// TIA Portal V19 export
FUNCTION_BLOCK "A0303_Sollevamento_FB"   // FB87, LAD
// stored: MemoryReserve 100, SetENOAutomatically false
   VAR_INPUT
      AreaInterface : "AreaInterface";
      ZSI : "udt_ZoneSafetyInterface";
      DSI_Feed_Testa : "udt_DeviceSafetyInterface";
      DSI_Feed_Coda : "udt_DeviceSafetyInterface";
      DataIn : Struct
         OP_Vai_A_Prelievo : Bool;
         OP_Vai_A_Deposito : Bool;
         LsSensor1_Carico : Bool;   // FTC 1 CONTROLLO POSIZIONE LIBERA IN CARICO
         LsSensor2_Carico : Bool;   // FTC 2 CONTROLLO POSIZIONE LIBERA IN CARICO
         LsSensor1_Scarico : Bool;   // FTC 1 CONTROLLO POSIZIONE LIBERA IN SCARICO
         LsSensor2_Scarico : Bool;   // FTC 2 CONTROLLO POSIZIONE LIBERA IN SCARICO
      END_STRUCT;
      CIn : Struct
         Manager : Struct
            EnableStopDoorOpeningReq : Bool;
            EnableStopInPhase : Bool;
            EnableStopProgrammed : Bool;
            Control_ON : Bool;
            CanMoveFreely : Bool;
            TargetPosition : LReal;
            Phase : Struct
               VAI_A_PRELIEVO : Bool;
               VAI_A_PRE_DEPOSITO : Bool;
               VAI_A_DEPOSITO : Bool;
            END_STRUCT;
         END_STRUCT;
         Trasporto : Struct
            IsMeasuring : Bool;
         END_STRUCT;
      END_STRUCT;
      Config : Struct
         Testa : Struct
            Ax : "Positioning_DOL_Machine_Config";
         END_STRUCT;
         Coda : Struct
            Ax : "Positioning_DOL_Machine_Config";
         END_STRUCT;
         DelayMissingCondition { ExternalAccessible := 'False'; ExternalVisible := 'False'; ExternalWritable := 'False'} : Time := T#0MS;
      END_STRUCT;
   END_VAR
   VAR_OUTPUT
      MachineInterface : "MachineInterface";
      COut : Struct
         Ax_Testa : "Positioning_DOL_Machine_COut";
         Ax_Coda : "Positioning_DOL_Machine_COut";
         Standstill : Bool;
         Minus_CheckNext : Bool;
         Plus_CheckNext : Bool;
         Minus_Running : Bool;
         Plus_Running : Bool;
      END_STRUCT;
   END_VAR
   VAR_IN_OUT
      Par : Struct
         Ax_Man : "Positioning_DOL_Machine_Par";
         Ax_Testa_Pers : "Positioning_DOL_Machine_Pers_Data";
         Ax_Coda_Pers : "Positioning_DOL_Machine_Pers_Data";
         Enc : Struct
            Testa : "PosFbk_RTN";
            Coda : "PosFbk_RTN";
         END_STRUCT;
      END_STRUCT;
      Par_Mach : Struct
         PosDeposito : LReal;
         OffsetPrelievo : LReal;
         ToleranceWindow : LReal;
      END_STRUCT;
   END_VAR
   VAR
      Alarm : Struct
         Testa : Struct
            Ax : "Positioning_DOL_Machine_Alr";
            Enc { S7_SetPoint := 'True'} : "PosFbk_Encoder_Alr";
         END_STRUCT;
         Coda : Struct
            Ax : "Positioning_DOL_Machine_Alr";
            Enc { S7_SetPoint := 'True'} : "PosFbk_Encoder_Alr";
         END_STRUCT;
         CheckBothAxMove : Bool;
      END_STRUCT;
      Warning : Struct
         Testa : Struct
            Ax { S7_SetPoint := 'True'} : "Positioning_DOL_Machine_Wng";
         END_STRUCT;
         Coda : Struct
            Ax { S7_SetPoint := 'True'} : "Positioning_DOL_Machine_Wng";
         END_STRUCT;
         MissingCnd : Struct
            OP_VAI_A_PRELIEVO : Bool;   // Mancanza consenso lavoro
            OP_VAI_A_DEPOSITO : Bool;   // Mancanza consenso lavoro
         END_STRUCT;
      END_STRUCT;
      HMI : Struct
         Selection : Struct
            Ax : Int;   // 0= BOTH ; 1= HEAD ; 2= TAIL
         END_STRUCT;
         Testa : Struct
            PbPreset : Bool;
            PresetValue : LReal;
         END_STRUCT;
         Coda : Struct
            PbPreset : Bool;
            PresetValue : LReal;
         END_STRUCT;
         PositionGraph : Int;
      END_STRUCT;
      Sts : Struct
         OP_CanMoveFreely : Bool;
         OP_Vai_A_Prelievo_Cnd : Bool;
         OP_Vai_A_Deposito_Cnd : Bool;
         OP_Vai_A_PreDeposito_Cnd : Bool;
         Coda_PermessoDaSynchOk : Bool;
         Testa_PermessoDaSynchOk : Bool;
      END_STRUCT;
      Ctrl : Struct
         Man : Struct
            OP_Vai_A_Prelievo : Bool;
            OP_Vai_A_Deposito : Bool;
         END_STRUCT;
         Aut : Struct
            OP_Vai_A_Prelievo : Bool;
            OP_Vai_A_Deposito : Bool;
            OP_Vai_A_PreDeposito : Bool;
         END_STRUCT;
         OP_Vai_A_Prelievo : Bool;
         OP_Vai_A_Deposito : Bool;
         OP_Vai_A_PreDeposito : Bool;
      END_STRUCT;
      Ax_Testa { S7_SetPoint := 'True'} : "Positioning_DOL_Machine_FB";
      Ax_Coda { S7_SetPoint := 'True'} : "Positioning_DOL_Machine_FB";
      Enc_Testa : "PosFbk_SickAFM60";
      Enc_Testa_ITF : "PosFbk_ITF";
      Enc_Coda : "PosFbk_SickAFM60";
      Enc_Coda_ITF : "PosFbk_ITF";
      AUX { ExternalAccessible := 'False'; ExternalVisible := 'False'; ExternalWritable := 'False'} : Struct
         OP_Vai_A_Prelievo : Bool;
         OP_Vai_A_Deposito : Bool;
      END_STRUCT;
      TON_OP_VAI_A_PRELIEVO_MissingCnd : IEC_TIMER;
      TON_OP_VAI_A_DEPOSITO_MissingCnd : IEC_TIMER;
      TON_CheckAxMove { S7_SetPoint := 'True'} : IEC_TIMER;
      TON_CheckAxis { S7_SetPoint := 'True'} : IEC_TIMER;
      CheckAxisSynch { S7_SetPoint := 'True'} : "CheckAxisSynch";
      Sts_PosAxis { S7_SetPoint := 'True'} : Int;
   END_VAR
   VAR_TEMP
      PE : Struct
         OP_Vai_A_Prelievo : Bool;
         OP_Vai_A_Deposito : Bool;
      END_STRUCT;
      PosDiff : LReal;
      Axis_Testa_Behind : Bool;
      Axis_Coda_Behind : Bool;
      ValueIn : LReal;
      X1 : LReal;
      X2 : LReal;
      Ret_Val : LReal;
   END_VAR
   VAR CONSTANT
      MaxDistance : LReal := 5.0;
      MinDistance : LReal := 0.5;   // soglia inferiore per isteresi
   END_VAR
   // Config.Testa.Ax.DelayMissingCondition := T#3S;
   // Config.Testa.Ax.CyclicOBTime_ms := 10.0;
   // Config.Testa.Ax.Ax.limitMinus := 0.0;
   // Config.Testa.Ax.Ax.limitPlus := 476.0;
   // Config.Testa.Ax.Ax.Backlash := 0.0;
   // Config.Testa.Ax.Ax.BacklashActivation := FALSE;
   // Config.Testa.Ax.Ax.ToleranceWindow := 0.1;
   // Config.Testa.Ax.Ax.ToleranceWindowDelay := T#100MS;
   // Config.Testa.Ax.Ax.PreCutOff := 0.0;
   // Config.Testa.Ax.Ax.PreEndLowSpeed := 0.0;
   // Config.Testa.Ax.Ax.PreEndMedSpeed := 0.0;
   // Config.Testa.Ax.Ax.ChangeDirectionDelay := T#0MS;
   // Config.Testa.Ax.Ax.StandstillVelocity := 0.5;
   // Config.Testa.Ax.Ax.StandStillDelay := T#100MS;
   // Config.Testa.Ax.Ax.HomingDirection := FALSE;
   // Config.Testa.Ax.Ax.RecallTime := 0.0;
   // Config.Testa.Ax.Ax.VelocityFilter_T := 10.0;
   // Config.Testa.Ax.Ax.VelocityMeasUnit := 2;
   // Config.Testa.Ax.Ax.PosFbkDisabled := FALSE;
   // Config.Testa.Ax.Ax.FbkCtrlDisabled := TRUE;
   // Config.Testa.Ax.Ax_UM2."m" := 1.0;
   // Config.Testa.Ax.Ax_UM2.q := 0.0;
   // Config.Testa.Ax.S120.SpeedMotor.ReferenceVelocity := 2000.0;
   // Config.Testa.Ax.S120.SpeedMotor.InvertDirection := FALSE;
   // Config.Testa.Ax.S120.PowerOffDelay := T#5S;
   // Config.Testa.Ax.S120.StandstillVelocity := 50.0;
   // Config.Testa.Ax.S120.AccTime := 0.25;
   // Config.Testa.Ax.S120.DecTime := 0.25;
   // Config.Testa.Ax.Fan.Presence := FALSE;
   // Config.Testa.Ax.Fan.DelayOff := T#10M;
   // Config.Testa.Ax.Brake_Presence := FALSE;
   // Config.Coda.Ax.DelayMissingCondition := T#3S;
   // Config.Coda.Ax.CyclicOBTime_ms := 10.0;
   // Config.Coda.Ax.Ax.limitMinus := 0.0;
   // Config.Coda.Ax.Ax.limitPlus := 476.0;
   // Config.Coda.Ax.Ax.Backlash := 0.0;
   // Config.Coda.Ax.Ax.BacklashActivation := FALSE;
   // Config.Coda.Ax.Ax.ToleranceWindow := 0.1;
   // Config.Coda.Ax.Ax.ToleranceWindowDelay := T#100MS;
   // Config.Coda.Ax.Ax.PreCutOff := 0.0;
   // Config.Coda.Ax.Ax.PreEndLowSpeed := 0.0;
   // Config.Coda.Ax.Ax.PreEndMedSpeed := 0.0;
   // Config.Coda.Ax.Ax.ChangeDirectionDelay := T#0MS;
   // Config.Coda.Ax.Ax.StandstillVelocity := 0.5;
   // Config.Coda.Ax.Ax.StandStillDelay := T#100MS;
   // Config.Coda.Ax.Ax.HomingDirection := FALSE;
   // Config.Coda.Ax.Ax.RecallTime := 0.0;
   // Config.Coda.Ax.Ax.VelocityFilter_T := 10.0;
   // Config.Coda.Ax.Ax.VelocityMeasUnit := 2;
   // Config.Coda.Ax.Ax.PosFbkDisabled := FALSE;
   // Config.Coda.Ax.Ax.FbkCtrlDisabled := TRUE;
   // Config.Coda.Ax.Ax_UM2."m" := 1.0;
   // Config.Coda.Ax.Ax_UM2.q := 0.0;
   // Config.Coda.Ax.S120.SpeedMotor.ReferenceVelocity := 2000.0;
   // Config.Coda.Ax.S120.SpeedMotor.InvertDirection := FALSE;
   // Config.Coda.Ax.S120.PowerOffDelay := T#5S;
   // Config.Coda.Ax.S120.StandstillVelocity := 50.0;
   // Config.Coda.Ax.S120.AccTime := 0.25;
   // Config.Coda.Ax.S120.DecTime := 0.25;
   // Config.Coda.Ax.Fan.Presence := FALSE;
   // Config.Coda.Ax.Fan.DelayOff := T#10M;
   // Config.Coda.Ax.Brake_Presence := FALSE;
   VAR_TEMP   // added for the SCL form of the ladder/FBD networks
      _w1 : Bool;
   END_VAR
BEGIN

REGION Network 1 (SCL): Reset allarmi
   IF #AreaInterface.RstAlarms THEN
       #Alarm.CheckBothAxMove := FALSE;
   END_IF;
END_REGION

REGION Network 2: <+>
END_REGION

REGION Network 3: <<<<<<<<<<<<<<<<<<< OPERAZIONI >>>>>>>>>>>>>>>>>>>>>>>>
END_REGION

REGION Network 4: Operazione può muoversi liberamente perchè non sposta nessun BEAM
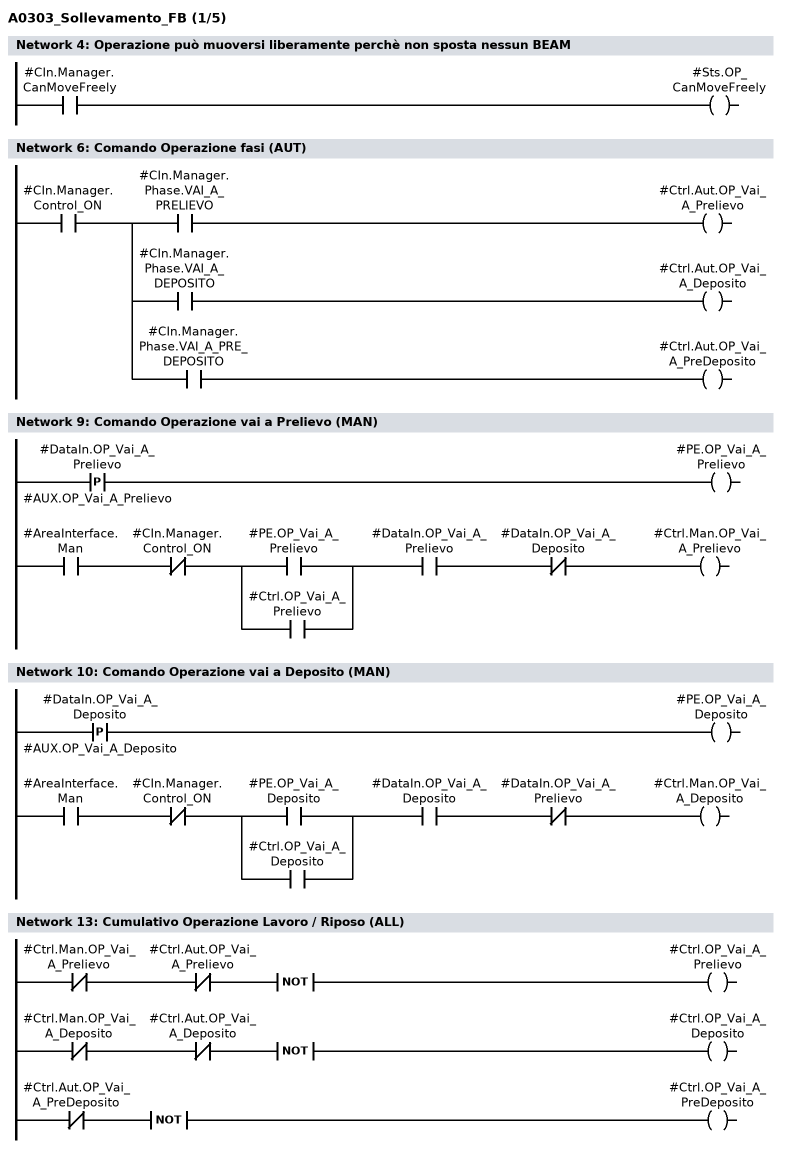
   RUNG wire#powerrail
      Contact( #CIn.Manager.CanMoveFreely )
      Coil( #Sts.OP_CanMoveFreely )
   END_RUNG
   // the same network as SCL:
   #Sts.OP_CanMoveFreely := #CIn.Manager.CanMoveFreely;
END_REGION

REGION Network 5: < OPERAZIONI AUTOMATICO >
END_REGION

REGION Network 6: Comando Operazione fasi (AUT)
   RUNG wire#powerrail
      Contact( #CIn.Manager.Control_ON )
      wire#w1
      Contact( #CIn.Manager.Phase.VAI_A_PRELIEVO )
      Coil( #Ctrl.Aut.OP_Vai_A_Prelievo )
   END_RUNG
   RUNG wire#w1
      Contact( #CIn.Manager.Phase.VAI_A_DEPOSITO )
      Coil( #Ctrl.Aut.OP_Vai_A_Deposito )
   END_RUNG
   RUNG wire#w1
      Contact( #CIn.Manager.Phase.VAI_A_PRE_DEPOSITO )
      Coil( #Ctrl.Aut.OP_Vai_A_PreDeposito )
   END_RUNG
   // the same network as SCL:
   #Ctrl.Aut.OP_Vai_A_Prelievo := #CIn.Manager.Control_ON AND #CIn.Manager.Phase.VAI_A_PRELIEVO;
   #Ctrl.Aut.OP_Vai_A_Deposito := #CIn.Manager.Control_ON AND #CIn.Manager.Phase.VAI_A_DEPOSITO;
   #Ctrl.Aut.OP_Vai_A_PreDeposito := #CIn.Manager.Control_ON AND #CIn.Manager.Phase.VAI_A_PRE_DEPOSITO;
END_REGION

REGION Network 7: <+>
END_REGION

REGION Network 8: < OPERAZIONI MANUALI >
END_REGION

REGION Network 9: Comando Operazione vai a Prelievo (MAN)
   RUNG wire#powerrail
      P_Contact(operand := #DataIn.OP_Vai_A_Prelievo, bit := #AUX.OP_Vai_A_Prelievo)
      Coil( #PE.OP_Vai_A_Prelievo )
   END_RUNG
   RUNG wire#powerrail
      Contact( #AreaInterface.Man )
      I_Contact( #CIn.Manager.Control_ON )
      wire#w1
      Contact( #PE.OP_Vai_A_Prelievo )
      wire#w2
      Contact( #DataIn.OP_Vai_A_Prelievo )
      I_Contact( #DataIn.OP_Vai_A_Deposito )
      Coil( #Ctrl.Man.OP_Vai_A_Prelievo )
   END_RUNG
   RUNG wire#w1
      Contact( #Ctrl.OP_Vai_A_Prelievo )
   END_RUNG wire#w2
   // the same network as SCL:
   #_w1 := #DataIn.OP_Vai_A_Prelievo AND NOT #AUX.OP_Vai_A_Prelievo;   // rising edge of #DataIn.OP_Vai_A_Prelievo
   #AUX.OP_Vai_A_Prelievo := #DataIn.OP_Vai_A_Prelievo;
   #PE.OP_Vai_A_Prelievo := #_w1;
   #Ctrl.Man.OP_Vai_A_Prelievo := #AreaInterface.Man AND NOT #CIn.Manager.Control_ON AND (#PE.OP_Vai_A_Prelievo OR #Ctrl.OP_Vai_A_Prelievo) AND #DataIn.OP_Vai_A_Prelievo AND NOT #DataIn.OP_Vai_A_Deposito;
END_REGION

REGION Network 10: Comando Operazione vai a Deposito (MAN)
   RUNG wire#powerrail
      P_Contact(operand := #DataIn.OP_Vai_A_Deposito, bit := #AUX.OP_Vai_A_Deposito)
      Coil( #PE.OP_Vai_A_Deposito )
   END_RUNG
   RUNG wire#powerrail
      Contact( #AreaInterface.Man )
      I_Contact( #CIn.Manager.Control_ON )
      wire#w1
      Contact( #PE.OP_Vai_A_Deposito )
      wire#w2
      Contact( #DataIn.OP_Vai_A_Deposito )
      I_Contact( #DataIn.OP_Vai_A_Prelievo )
      Coil( #Ctrl.Man.OP_Vai_A_Deposito )
   END_RUNG
   RUNG wire#w1
      Contact( #Ctrl.OP_Vai_A_Deposito )
   END_RUNG wire#w2
   // the same network as SCL:
   #_w1 := #DataIn.OP_Vai_A_Deposito AND NOT #AUX.OP_Vai_A_Deposito;   // rising edge of #DataIn.OP_Vai_A_Deposito
   #AUX.OP_Vai_A_Deposito := #DataIn.OP_Vai_A_Deposito;
   #PE.OP_Vai_A_Deposito := #_w1;
   #Ctrl.Man.OP_Vai_A_Deposito := #AreaInterface.Man AND NOT #CIn.Manager.Control_ON AND (#PE.OP_Vai_A_Deposito OR #Ctrl.OP_Vai_A_Deposito) AND #DataIn.OP_Vai_A_Deposito AND NOT #DataIn.OP_Vai_A_Prelievo;
END_REGION

REGION Network 11: <+>
END_REGION

REGION Network 12: < CUMULATIVO OPERAZIONI >
END_REGION

REGION Network 13: Cumulativo Operazione Lavoro / Riposo (ALL)
   RUNG wire#powerrail
      I_Contact( #Ctrl.Man.OP_Vai_A_Prelievo )
      I_Contact( #Ctrl.Aut.OP_Vai_A_Prelievo )
      Not()
      Coil( #Ctrl.OP_Vai_A_Prelievo )
   END_RUNG
   RUNG wire#powerrail
      I_Contact( #Ctrl.Man.OP_Vai_A_Deposito )
      I_Contact( #Ctrl.Aut.OP_Vai_A_Deposito )
      Not()
      Coil( #Ctrl.OP_Vai_A_Deposito )
   END_RUNG
   RUNG wire#powerrail
      I_Contact( #Ctrl.Aut.OP_Vai_A_PreDeposito )
      Not()
      Coil( #Ctrl.OP_Vai_A_PreDeposito )
   END_RUNG
   // the same network as SCL:
   #Ctrl.OP_Vai_A_Prelievo := NOT (NOT #Ctrl.Man.OP_Vai_A_Prelievo AND NOT #Ctrl.Aut.OP_Vai_A_Prelievo);
   #Ctrl.OP_Vai_A_Deposito := NOT (NOT #Ctrl.Man.OP_Vai_A_Deposito AND NOT #Ctrl.Aut.OP_Vai_A_Deposito);
   #Ctrl.OP_Vai_A_PreDeposito := NOT (NOT #Ctrl.Aut.OP_Vai_A_PreDeposito);
END_REGION

REGION Network 14: <+>
END_REGION

REGION Network 15: < CONDIZIONI MOVIMENTO >
END_REGION

REGION Network 16: Condizioni movimento Operazione a Lavoro / Riposo
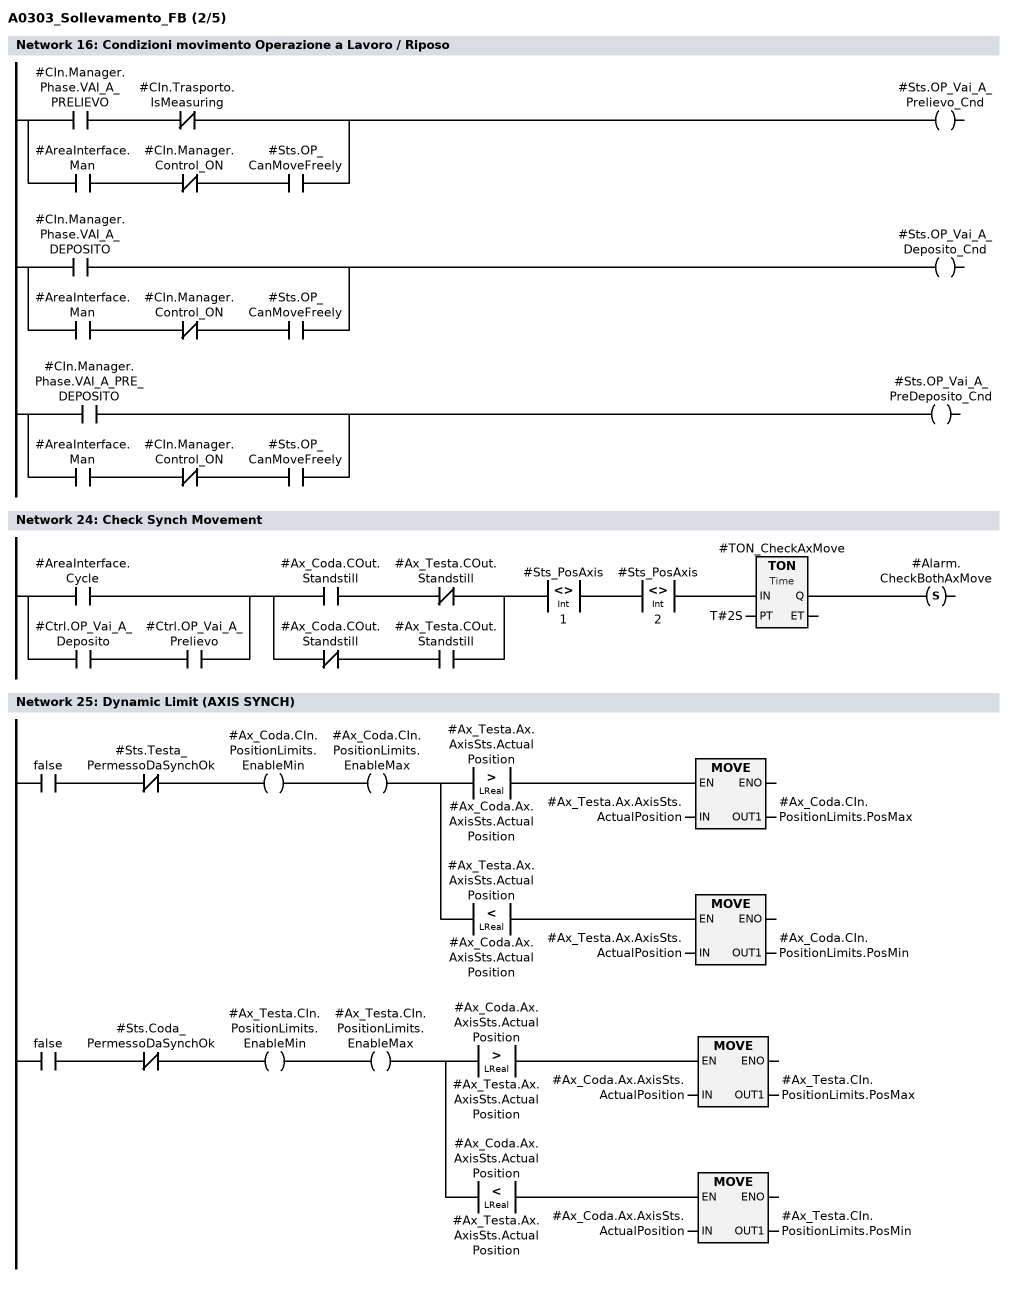
   RUNG wire#powerrail
      Contact( #CIn.Manager.Phase.VAI_A_PRELIEVO )
      I_Contact( #CIn.Trasporto.IsMeasuring )
      wire#w1
      Coil( #Sts.OP_Vai_A_Prelievo_Cnd )
   END_RUNG
   RUNG wire#powerrail
      Contact( #AreaInterface.Man )
      I_Contact( #CIn.Manager.Control_ON )
      Contact( #Sts.OP_CanMoveFreely )
   END_RUNG wire#w1
   RUNG wire#powerrail
      Contact( #CIn.Manager.Phase.VAI_A_DEPOSITO )
      wire#w2
      Coil( #Sts.OP_Vai_A_Deposito_Cnd )
   END_RUNG
   RUNG wire#powerrail
      Contact( #AreaInterface.Man )
      I_Contact( #CIn.Manager.Control_ON )
      Contact( #Sts.OP_CanMoveFreely )
   END_RUNG wire#w2
   RUNG wire#powerrail
      Contact( #CIn.Manager.Phase.VAI_A_PRE_DEPOSITO )
      wire#w3
      Coil( #Sts.OP_Vai_A_PreDeposito_Cnd )
   END_RUNG
   RUNG wire#powerrail
      Contact( #AreaInterface.Man )
      I_Contact( #CIn.Manager.Control_ON )
      Contact( #Sts.OP_CanMoveFreely )
   END_RUNG wire#w3
   // the same network as SCL:
   #Sts.OP_Vai_A_Prelievo_Cnd := (#CIn.Manager.Phase.VAI_A_PRELIEVO AND NOT #CIn.Trasporto.IsMeasuring) OR (#AreaInterface.Man AND NOT #CIn.Manager.Control_ON AND #Sts.OP_CanMoveFreely);
   #Sts.OP_Vai_A_Deposito_Cnd := #CIn.Manager.Phase.VAI_A_DEPOSITO OR (#AreaInterface.Man AND NOT #CIn.Manager.Control_ON AND #Sts.OP_CanMoveFreely);
   #Sts.OP_Vai_A_PreDeposito_Cnd := #CIn.Manager.Phase.VAI_A_PRE_DEPOSITO OR (#AreaInterface.Man AND NOT #CIn.Manager.Control_ON AND #Sts.OP_CanMoveFreely);
END_REGION

REGION Network 17: <+>
END_REGION

REGION Network 18: <<<<<<<<<<<<<<<<<<< SEQUENZA COMANDI >>>>>>>>>>>>>>>>>>>>>>>>
END_REGION

REGION Network 19 (SCL): Sincronizzazione tra asse testa e asse coda
   #CheckAxisSynch(Ax1_Pos:=#Ax_Testa.Sts.ActualPosition,
                            Ax2_Pos:=#Ax_Coda.Sts.ActualPosition,
                            TargetPos:=#Ax_Testa.Ctrl.Pos,
                            MaxDistance:=#MaxDistance,
                            MinDistance:=#MinDistance,
                            Ax1_SynchOk=> #Sts.Testa_PermessoDaSynchOk,
                            Ax2_SynchOk=> #Sts.Coda_PermessoDaSynchOk);
END_REGION

REGION Network 20: <+>
END_REGION

REGION Network 21 (SCL): CIn Abilitazioni Stop Manager
   // CIn Manager Stop per richiesta apertura safety
   // 
   #Ax_Testa.CIn.Manager.EnableStopDoorOpeningReq := #Ax_Coda.CIn.Manager.EnableStopDoorOpeningReq := #CIn.Manager.EnableStopDoorOpeningReq;

   // CIn Manager Stop in fase delle macchine precedenti
   // 
   #Ax_Testa.CIn.Manager.EnableStopInPhase := #Ax_Coda.CIn.Manager.EnableStopInPhase := #CIn.Manager.EnableStopInPhase;

   // CIn Manager Stop programmato configurabile a piacere
   // 
   #Ax_Testa.CIn.Manager.EnableStopProgrammed := #Ax_Coda.CIn.Manager.EnableStopProgrammed := #CIn.Manager.EnableStopProgrammed;
END_REGION

REGION Network 22 (SCL): Cin Manager (Esecuzione sequenza comandi)
   //CTRL ON
   #Ax_Testa.CIn.Manager.Control_ON := #Ax_Coda.CIn.Manager.Control_ON := #Ctrl.OP_Vai_A_Deposito  OR #Ctrl.OP_Vai_A_Prelievo OR #Ctrl.OP_Vai_A_PreDeposito ;

   #Ax_Testa.CIn.Manager.Speed := #Ax_Coda.CIn.Manager.Speed := 100;

   #TON_CheckAxis.TON(IN := #Sts_PosAxis = 2  OR #Sts_PosAxis = 3,
                      PT := T#0.5S);


   //Power On Assi
   #Ax_Coda.CIn.ExternalPowerOn := #Ax_Testa.CIn.ExternalPowerOn := #Ctrl.OP_Vai_A_Prelievo OR #Ctrl.OP_Vai_A_Deposito OR #Ctrl.OP_Vai_A_PreDeposito;


   IF #Sts_PosAxis = 3 AND ABS(#Ax_Testa.Sts.ActualPosition - #Ax_Coda.Sts.ActualPosition) > #MaxDistance THEN
       #Sts_PosAxis := 0;
   END_IF;

   IF NOT #Ctrl.OP_Vai_A_Deposito AND NOT #Ctrl.OP_Vai_A_Prelievo AND NOT #Ctrl.OP_Vai_A_PreDeposito THEN
       #Sts_PosAxis := 0;
   END_IF;

   IF #Sts_PosAxis = 0 THEN

       #Ax_Testa.CIn.Manager.MoveToPos := #Ax_Coda.CIn.Manager.MoveToPos := FALSE;

       IF #Ctrl.OP_Vai_A_Deposito OR #Ctrl.OP_Vai_A_Prelievo OR #Ctrl.OP_Vai_A_PreDeposito THEN
           IF ABS(#Ax_Testa.Sts.ActualPosition - #Ax_Coda.Sts.ActualPosition) > #MaxDistance THEN

               #Ax_Testa.CIn.Manager.Pos := #Ax_Coda.Sts.ActualPosition;
               #Ax_Coda.CIn.Manager.Pos := #Ax_Coda.Sts.ActualPosition;
               #Ax_Coda.CIn.Manager.MoveToPos := TRUE;
               #Ax_Testa.CIn.Manager.MoveToPos := TRUE;
               #Ax_Coda.CIn.Manager.Speed := #Ax_Testa.CIn.Manager.Speed :=50;


               #Sts_PosAxis := 1;
           ELSE
               #Sts_PosAxis := 3;
           END_IF;

       END_IF;
   END_IF;

   IF #Sts_PosAxis = 1 THEN

       IF ABS(#Ax_Testa.Sts.ActualPosition - #Ax_Coda.Sts.ActualPosition) < #MinDistance THEN
           #Ax_Testa.CIn.Manager.MoveToPos := FALSE;
           #Ax_Coda.CIn.Manager.MoveToPos := FALSE;

           #Sts_PosAxis := 2;

       END_IF;

   END_IF;



   IF #Sts_PosAxis = 2 THEN


       #Ax_Testa.CIn.Manager.MoveToPos := FALSE;
       #Ax_Coda.CIn.Manager.MoveToPos := FALSE;

       IF #Ax_Coda.COut.Standstill AND #Ax_Testa.COut.Standstill AND #TON_CheckAxis.Q THEN

           #Sts_PosAxis := 3;
       END_IF;

   END_IF;


   IF #Sts_PosAxis = 3 AND NOT #Alarm.CheckBothAxMove THEN

       #Ax_Testa.CIn.Manager.MoveToPos := FALSE;
       #Ax_Coda.CIn.Manager.MoveToPos := FALSE;


       IF #Ctrl.OP_Vai_A_Prelievo AND #Sts.OP_Vai_A_Prelievo_Cnd THEN

           //Power On Assi
           #Ax_Coda.CIn.ExternalPowerOn := #Ax_Testa.CIn.ExternalPowerOn := TRUE;

           // Sollevatore in posizione di Prelievo
           #Ax_Coda.CIn.Manager.Pos := #Ax_Testa.CIn.Manager.Pos := #CIn.Manager.TargetPosition;
           #Ax_Coda.CIn.Manager.Speed := #Ax_Testa.CIn.Manager.Speed := 100; //SARA DA GESTIRE
           #Ax_Testa.CIn.Manager.MoveToPos := NOT (#Ax_Testa.COut.InPosition AND (#Ax_Testa.COut.ActualTargetPos = #CIn.Manager.TargetPosition)) AND #Ax_Testa.S120.Sts.AxisEnabled AND #Ax_Coda.S120.Sts.AxisEnabled AND #TON_CheckAxis.Q;
           #Ax_Coda.CIn.Manager.MoveToPos := NOT (#Ax_Coda.COut.InPosition AND (#Ax_Coda.COut.ActualTargetPos = #CIn.Manager.TargetPosition)) AND #Ax_Testa.S120.Sts.AxisEnabled AND #Ax_Coda.S120.Sts.AxisEnabled AND #TON_CheckAxis.Q;



       ELSIF #Ctrl.OP_Vai_A_Deposito AND #Sts.OP_Vai_A_Deposito_Cnd THEN

           //Power On Assi
           #Ax_Coda.CIn.ExternalPowerOn := #Ax_Testa.CIn.ExternalPowerOn := TRUE;

           // Sollevatore in posizione di Deposito
           #Ax_Coda.CIn.Manager.Pos := #Ax_Testa.CIn.Manager.Pos := #Par_Mach.PosDeposito;
           #Ax_Coda.CIn.Manager.Speed := #Ax_Testa.CIn.Manager.Speed := 100.0; //SARA DA GESTIRE
           #Ax_Testa.CIn.Manager.MoveToPos := NOT (#Ax_Testa.COut.InPosition AND (#Ax_Testa.COut.ActualTargetPos = #Par_Mach.PosDeposito)) AND #Ax_Testa.S120.Sts.AxisEnabled AND #Ax_Coda.S120.Sts.AxisEnabled AND #TON_CheckAxis.Q;
           #Ax_Coda.CIn.Manager.MoveToPos := NOT (#Ax_Coda.COut.InPosition AND (#Ax_Coda.COut.ActualTargetPos = #Par_Mach.PosDeposito)) AND #Ax_Testa.S120.Sts.AxisEnabled AND #Ax_Coda.S120.Sts.AxisEnabled AND #TON_CheckAxis.Q;

       ELSIF #Ctrl.OP_Vai_A_PreDeposito AND #Sts.OP_Vai_A_PreDeposito_Cnd THEN

           //Power On Assi
           #Ax_Coda.CIn.ExternalPowerOn := #Ax_Testa.CIn.ExternalPowerOn := TRUE;

           // Sollevatore in posizione di Deposito
           #Ax_Coda.CIn.Manager.Pos := #Ax_Testa.CIn.Manager.Pos := #Par_Mach.PosDeposito - 10;
           #Ax_Coda.CIn.Manager.Speed := #Ax_Testa.CIn.Manager.Speed := 100.0; //SARA DA GESTIRE
           #Ax_Testa.CIn.Manager.MoveToPos := NOT (#Ax_Testa.COut.InPosition AND (#Ax_Testa.COut.ActualTargetPos = #Par_Mach.PosDeposito - 10)) AND #Ax_Testa.S120.Sts.AxisEnabled AND #Ax_Coda.S120.Sts.AxisEnabled AND #TON_CheckAxis.Q;
           #Ax_Coda.CIn.Manager.MoveToPos := NOT (#Ax_Coda.COut.InPosition AND (#Ax_Coda.COut.ActualTargetPos = #Par_Mach.PosDeposito - 10)) AND #Ax_Testa.S120.Sts.AxisEnabled AND #Ax_Coda.S120.Sts.AxisEnabled AND #TON_CheckAxis.Q;

       END_IF;
   END_IF;

   IF NOT #Ctrl.OP_Vai_A_Deposito AND NOT #Ctrl.OP_Vai_A_PreDeposito AND NOT #Ctrl.OP_Vai_A_Prelievo THEN
       // Reset Cmd
       #Ax_Testa.CIn.Manager.Minus := FALSE;
       #Ax_Coda.CIn.Manager.Minus := FALSE;
       #Ax_Testa.CIn.Manager.Plus := FALSE;
       #Ax_Coda.CIn.Manager.Plus := FALSE;
       #Ax_Coda.CIn.Manager.MoveToPos := FALSE;
       #Ax_Testa.CIn.Manager.MoveToPos := FALSE;
       #Ax_Coda.CIn.ExternalPowerOn := #Ax_Testa.CIn.ExternalPowerOn := FALSE;

   END_IF;
END_REGION

REGION Network 23: <+>
END_REGION

REGION Network 24: Check Synch Movement
   RUNG wire#powerrail
      Contact( #AreaInterface.Cycle )
      wire#w1
      Contact( #Ax_Coda.COut.Standstill )
      I_Contact( #Ax_Testa.COut.Standstill )
      wire#w2
      { S7_Templates := "SrcType := Int" } NE_Contact(in1 := #Sts_PosAxis, in2 := 1)
      { S7_Templates := "SrcType := Int" } NE_Contact(in1 := #Sts_PosAxis, in2 := 2)
      { S7_Templates := "time_type := Time" } #TON_CheckAxMove.TON(pt := T#2S, et =>)
      S_Coil( #Alarm.CheckBothAxMove )
   END_RUNG
   RUNG wire#powerrail
      Contact( #Ctrl.OP_Vai_A_Deposito )
      Contact( #Ctrl.OP_Vai_A_Prelievo )
   END_RUNG wire#w1
   RUNG wire#w1
      I_Contact( #Ax_Coda.COut.Standstill )
      Contact( #Ax_Testa.COut.Standstill )
   END_RUNG wire#w2
   // the same network as SCL:
   #TON_CheckAxMove.TON(IN := (#AreaInterface.Cycle OR (#Ctrl.OP_Vai_A_Deposito AND #Ctrl.OP_Vai_A_Prelievo)) AND ((#Ax_Coda.COut.Standstill AND NOT #Ax_Testa.COut.Standstill) OR (NOT #Ax_Coda.COut.Standstill AND #Ax_Testa.COut.Standstill)) AND (#Sts_PosAxis <> 1) AND (#Sts_PosAxis <> 2),
                        PT := T#2S);
   IF #TON_CheckAxMove.Q THEN #Alarm.CheckBothAxMove := TRUE; END_IF;
END_REGION

REGION Network 25: Dynamic Limit (AXIS SYNCH)
   RUNG wire#powerrail
      Contact( false )
      I_Contact( #Sts.Testa_PermessoDaSynchOk )
      Coil( #Ax_Coda.CIn.PositionLimits.EnableMin )
      Coil( #Ax_Coda.CIn.PositionLimits.EnableMax )
      wire#w1
      { S7_Templates := "SrcType := LReal" } GT_Contact(in1 := #Ax_Testa.Ax.AxisSts.ActualPosition, in2 := #Ax_Coda.Ax.AxisSts.ActualPosition)
      Move(in := #Ax_Testa.Ax.AxisSts.ActualPosition, out1 => #Ax_Coda.CIn.PositionLimits.PosMax)
   END_RUNG
   RUNG wire#w1
      { S7_Templates := "SrcType := LReal" } LT_Contact(in1 := #Ax_Testa.Ax.AxisSts.ActualPosition, in2 := #Ax_Coda.Ax.AxisSts.ActualPosition)
      Move(in := #Ax_Testa.Ax.AxisSts.ActualPosition, out1 => #Ax_Coda.CIn.PositionLimits.PosMin)
   END_RUNG
   RUNG wire#powerrail
      Contact( false )
      I_Contact( #Sts.Coda_PermessoDaSynchOk )
      Coil( #Ax_Testa.CIn.PositionLimits.EnableMin )
      Coil( #Ax_Testa.CIn.PositionLimits.EnableMax )
      wire#w2
      { S7_Templates := "SrcType := LReal" } GT_Contact(in1 := #Ax_Coda.Ax.AxisSts.ActualPosition, in2 := #Ax_Testa.Ax.AxisSts.ActualPosition)
      Move(in := #Ax_Coda.Ax.AxisSts.ActualPosition, out1 => #Ax_Testa.CIn.PositionLimits.PosMax)
   END_RUNG
   RUNG wire#w2
      { S7_Templates := "SrcType := LReal" } LT_Contact(in1 := #Ax_Coda.Ax.AxisSts.ActualPosition, in2 := #Ax_Testa.Ax.AxisSts.ActualPosition)
      Move(in := #Ax_Coda.Ax.AxisSts.ActualPosition, out1 => #Ax_Testa.CIn.PositionLimits.PosMin)
   END_RUNG
   // the same network as SCL:
   #Ax_Coda.CIn.PositionLimits.EnableMin := false AND NOT #Sts.Testa_PermessoDaSynchOk;
   #Ax_Coda.CIn.PositionLimits.EnableMax := #Ax_Coda.CIn.PositionLimits.EnableMin;
   IF #Ax_Coda.CIn.PositionLimits.EnableMin AND (#Ax_Testa.Ax.AxisSts.ActualPosition > #Ax_Coda.Ax.AxisSts.ActualPosition) THEN
       #Ax_Coda.CIn.PositionLimits.PosMax := #Ax_Testa.Ax.AxisSts.ActualPosition;
   END_IF;
   IF #Ax_Coda.CIn.PositionLimits.EnableMin AND (#Ax_Testa.Ax.AxisSts.ActualPosition < #Ax_Coda.Ax.AxisSts.ActualPosition) THEN
       #Ax_Coda.CIn.PositionLimits.PosMin := #Ax_Testa.Ax.AxisSts.ActualPosition;
   END_IF;
   #Ax_Testa.CIn.PositionLimits.EnableMin := false AND NOT #Sts.Coda_PermessoDaSynchOk;
   #Ax_Testa.CIn.PositionLimits.EnableMax := #Ax_Testa.CIn.PositionLimits.EnableMin;
   IF #Ax_Testa.CIn.PositionLimits.EnableMin AND (#Ax_Coda.Ax.AxisSts.ActualPosition > #Ax_Testa.Ax.AxisSts.ActualPosition) THEN
       #Ax_Testa.CIn.PositionLimits.PosMax := #Ax_Coda.Ax.AxisSts.ActualPosition;
   END_IF;
   IF #Ax_Testa.CIn.PositionLimits.EnableMin AND (#Ax_Coda.Ax.AxisSts.ActualPosition < #Ax_Testa.Ax.AxisSts.ActualPosition) THEN
       #Ax_Testa.CIn.PositionLimits.PosMin := #Ax_Coda.Ax.AxisSts.ActualPosition;
   END_IF;
END_REGION

REGION Network 26: <<<<<<<<<<<<<<<<<<<<<<<<<<<<<<<<<< LATO TESTA >>>>>>>>>>>>>>>>>>>>>>>>>>>>>>>>>>>>>>>
END_REGION

REGION Network 27: <<< ASSE MOVIMENTO >>>
END_REGION

REGION Network 28: [Ax] - Cin Ext Enable
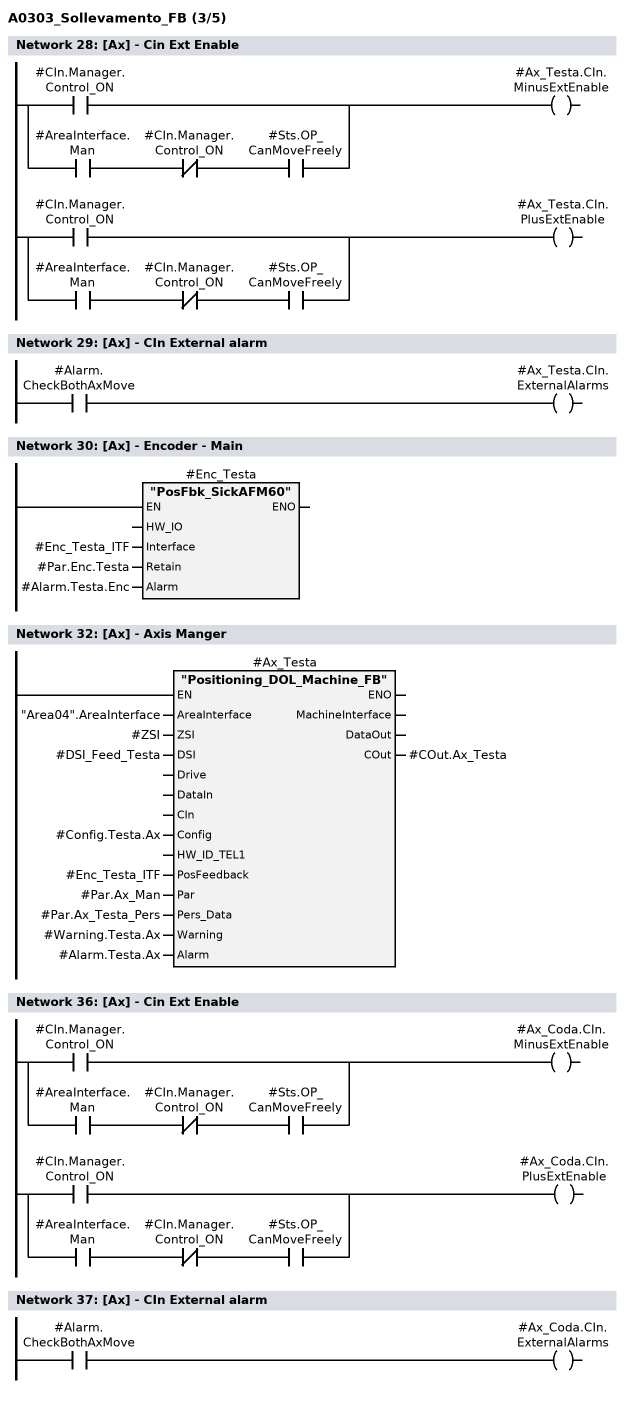
   RUNG wire#powerrail
      Contact( #CIn.Manager.Control_ON )
      wire#w1
      Coil( #Ax_Testa.CIn.MinusExtEnable )
   END_RUNG
   RUNG wire#powerrail
      Contact( #AreaInterface.Man )
      I_Contact( #CIn.Manager.Control_ON )
      Contact( #Sts.OP_CanMoveFreely )
   END_RUNG wire#w1
   RUNG wire#powerrail
      Contact( #CIn.Manager.Control_ON )
      wire#w2
      Coil( #Ax_Testa.CIn.PlusExtEnable )
   END_RUNG
   RUNG wire#powerrail
      Contact( #AreaInterface.Man )
      I_Contact( #CIn.Manager.Control_ON )
      Contact( #Sts.OP_CanMoveFreely )
   END_RUNG wire#w2
   // the same network as SCL:
   #Ax_Testa.CIn.MinusExtEnable := #CIn.Manager.Control_ON OR (#AreaInterface.Man AND NOT #CIn.Manager.Control_ON AND #Sts.OP_CanMoveFreely);
   #Ax_Testa.CIn.PlusExtEnable := #CIn.Manager.Control_ON OR (#AreaInterface.Man AND NOT #CIn.Manager.Control_ON AND #Sts.OP_CanMoveFreely);
END_REGION

REGION Network 29: [Ax] - CIn External alarm
   RUNG wire#powerrail
      Contact( #Alarm.CheckBothAxMove )
      Coil( #Ax_Testa.CIn.ExternalAlarms )
   END_RUNG
   // the same network as SCL:
   #Ax_Testa.CIn.ExternalAlarms := #Alarm.CheckBothAxMove;
END_REGION

REGION Network 30: [Ax] - Encoder - Main
   RUNG wire#powerrail
      #Enc_Testa(HW_IO :=, Interface := #Enc_Testa_ITF, Retain := #Par.Enc.Testa, Alarm := #Alarm.Testa.Enc)
   END_RUNG
   // the same network as SCL:
   #Enc_Testa(Interface := #Enc_Testa_ITF, Retain := #Par.Enc.Testa, Alarm := #Alarm.Testa.Enc);   // "PosFbk_SickAFM60"
END_REGION

REGION Network 31 (SCL): HMI preset position
   #Ax_Testa.HMI.B_Preset := #HMI.Testa.PbPreset;

   #Ax_Testa.HMI.PresetPosition := #HMI.Testa.PresetValue;
END_REGION

REGION Network 32: [Ax] - Axis Manger
   RUNG wire#powerrail
      #Ax_Testa(AreaInterface := "Area04".AreaInterface, ZSI := #ZSI, DSI := #DSI_Feed_Testa, Drive :=, DataIn :=, CIn :=, Config := #Config.Testa.Ax, HW_ID_TEL1 :=, PosFeedback := #Enc_Testa_ITF, Par := #Par.Ax_Man, Pers_Data := #Par.Ax_Testa_Pers, Warning := #Warning.Testa.Ax, Alarm := #Alarm.Testa.Ax, MachineInterface =>, DataOut =>, COut => #COut.Ax_Testa)
   END_RUNG
   // the same network as SCL:
   #Ax_Testa(AreaInterface := "Area04".AreaInterface,   // "Positioning_DOL_Machine_FB"
             ZSI := #ZSI,
             DSI := #DSI_Feed_Testa,
             Config := #Config.Testa.Ax,
             PosFeedback := #Enc_Testa_ITF,
             Par := #Par.Ax_Man,
             Pers_Data := #Par.Ax_Testa_Pers,
             Warning := #Warning.Testa.Ax,
             Alarm := #Alarm.Testa.Ax,
             COut => #COut.Ax_Testa);
END_REGION

REGION Network 34: <<<<<<<<<<<<<<<<<<<<<<<<<<<<<<<<<< LATO CODA >>>>>>>>>>>>>>>>>>>>>>>>>>>>>>>>>>>>>>>
END_REGION

REGION Network 35: <<< ASSE MOVIMENTO >>>
END_REGION

REGION Network 36: [Ax] - Cin Ext Enable
   RUNG wire#powerrail
      Contact( #CIn.Manager.Control_ON )
      wire#w1
      Coil( #Ax_Coda.CIn.MinusExtEnable )
   END_RUNG
   RUNG wire#powerrail
      Contact( #AreaInterface.Man )
      I_Contact( #CIn.Manager.Control_ON )
      Contact( #Sts.OP_CanMoveFreely )
   END_RUNG wire#w1
   RUNG wire#powerrail
      Contact( #CIn.Manager.Control_ON )
      wire#w2
      Coil( #Ax_Coda.CIn.PlusExtEnable )
   END_RUNG
   RUNG wire#powerrail
      Contact( #AreaInterface.Man )
      I_Contact( #CIn.Manager.Control_ON )
      Contact( #Sts.OP_CanMoveFreely )
   END_RUNG wire#w2
   // the same network as SCL:
   #Ax_Coda.CIn.MinusExtEnable := #CIn.Manager.Control_ON OR (#AreaInterface.Man AND NOT #CIn.Manager.Control_ON AND #Sts.OP_CanMoveFreely);
   #Ax_Coda.CIn.PlusExtEnable := #CIn.Manager.Control_ON OR (#AreaInterface.Man AND NOT #CIn.Manager.Control_ON AND #Sts.OP_CanMoveFreely);
END_REGION

REGION Network 37: [Ax] - CIn External alarm
   RUNG wire#powerrail
      Contact( #Alarm.CheckBothAxMove )
      Coil( #Ax_Coda.CIn.ExternalAlarms )
   END_RUNG
   // the same network as SCL:
   #Ax_Coda.CIn.ExternalAlarms := #Alarm.CheckBothAxMove;
END_REGION

REGION Network 38: [Ax] - Encoder - Main
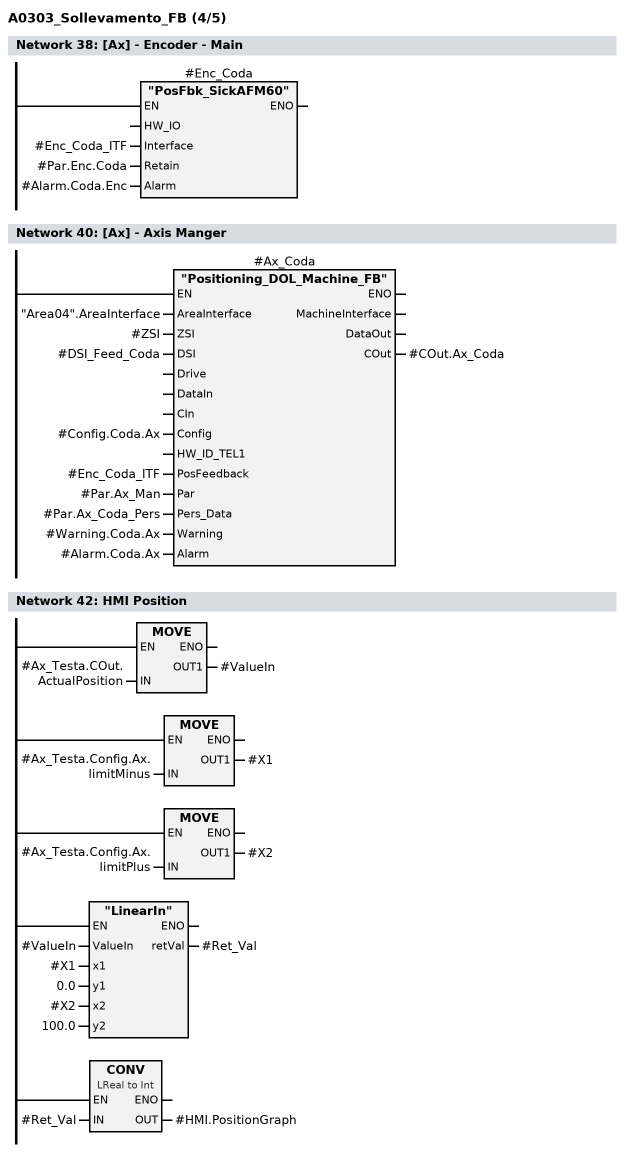
   RUNG wire#powerrail
      #Enc_Coda(HW_IO :=, Interface := #Enc_Coda_ITF, Retain := #Par.Enc.Coda, Alarm := #Alarm.Coda.Enc)
   END_RUNG
   // the same network as SCL:
   #Enc_Coda(Interface := #Enc_Coda_ITF, Retain := #Par.Enc.Coda, Alarm := #Alarm.Coda.Enc);   // "PosFbk_SickAFM60"
END_REGION

REGION Network 39 (SCL): HMI preset position
   #Ax_Coda.HMI.B_Preset := #HMI.Coda.PbPreset;

   #Ax_Coda.HMI.PresetPosition := #HMI.Coda.PresetValue;
END_REGION

REGION Network 40: [Ax] - Axis Manger
   RUNG wire#powerrail
      #Ax_Coda(AreaInterface := "Area04".AreaInterface, ZSI := #ZSI, DSI := #DSI_Feed_Coda, Drive :=, DataIn :=, CIn :=, Config := #Config.Coda.Ax, HW_ID_TEL1 :=, PosFeedback := #Enc_Coda_ITF, Par := #Par.Ax_Man, Pers_Data := #Par.Ax_Coda_Pers, Warning := #Warning.Coda.Ax, Alarm := #Alarm.Coda.Ax, MachineInterface =>, DataOut =>, COut => #COut.Ax_Coda)
   END_RUNG
   // the same network as SCL:
   #Ax_Coda(AreaInterface := "Area04".AreaInterface,   // "Positioning_DOL_Machine_FB"
            ZSI := #ZSI,
            DSI := #DSI_Feed_Coda,
            Config := #Config.Coda.Ax,
            PosFeedback := #Enc_Coda_ITF,
            Par := #Par.Ax_Man,
            Pers_Data := #Par.Ax_Coda_Pers,
            Warning := #Warning.Coda.Ax,
            Alarm := #Alarm.Coda.Ax,
            COut => #COut.Ax_Coda);
END_REGION

REGION Network 41: <+>
END_REGION

REGION Network 42: HMI Position
   RUNG wire#powerrail
      Move(in := #Ax_Testa.COut.ActualPosition, out1 => #ValueIn)
   END_RUNG
   RUNG wire#powerrail
      Move(in := #Ax_Testa.Config.Ax.limitMinus, out1 => #X1)
   END_RUNG
   RUNG wire#powerrail
      Move(in := #Ax_Testa.Config.Ax.limitPlus, out1 => #X2)
   END_RUNG
   RUNG wire#powerrail
      "LinearIn"(ValueIn := #ValueIn, x1 := #X1, y1 := 0.0, x2 := #X2, y2 := 100.0, retVal => #Ret_Val)
   END_RUNG
   RUNG wire#powerrail
      { S7_Templates := "[SrcType := LReal, DestType := Int]" } Convert(in := #Ret_Val, out => #HMI.PositionGraph)
   END_RUNG
   // the same network as SCL:
   #ValueIn := #Ax_Testa.COut.ActualPosition;
   #X1 := #Ax_Testa.Config.Ax.limitMinus;
   #X2 := #Ax_Testa.Config.Ax.limitPlus;
   "LinearIn"(ValueIn := #ValueIn, x1 := #X1, y1 := 0.0, x2 := #X2, y2 := 100.0, retVal => #Ret_Val);
   #HMI.PositionGraph := LREAL_TO_INT(#Ret_Val);
END_REGION

REGION Network 43: [Ax] - COut
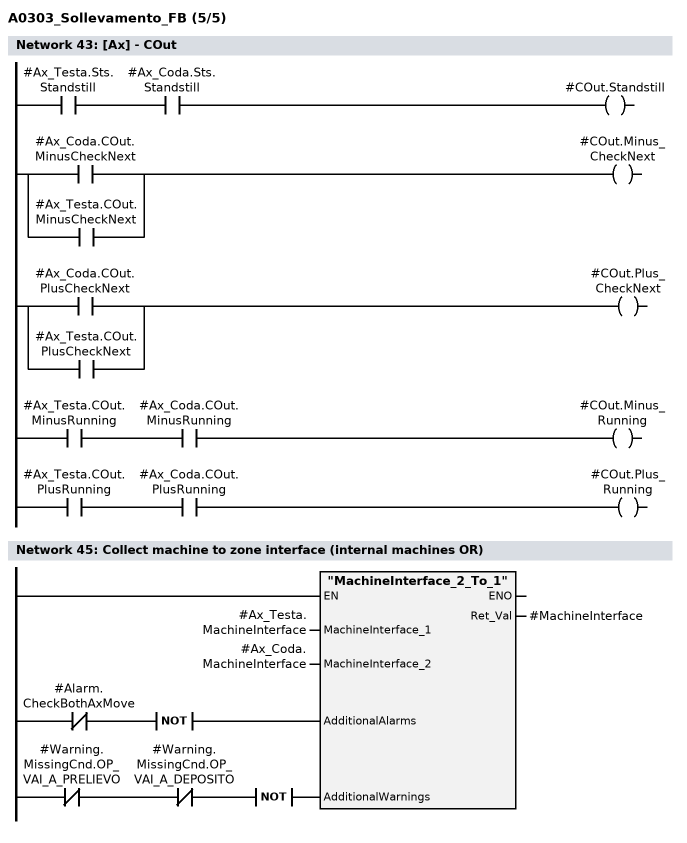
   RUNG wire#powerrail
      Contact( #Ax_Testa.Sts.Standstill )
      Contact( #Ax_Coda.Sts.Standstill )
      Coil( #COut.Standstill )
   END_RUNG
   RUNG wire#powerrail
      Contact( #Ax_Coda.COut.MinusCheckNext )
      wire#w1
      Coil( #COut.Minus_CheckNext )
   END_RUNG
   RUNG wire#powerrail
      Contact( #Ax_Testa.COut.MinusCheckNext )
   END_RUNG wire#w1
   RUNG wire#powerrail
      Contact( #Ax_Coda.COut.PlusCheckNext )
      wire#w2
      Coil( #COut.Plus_CheckNext )
   END_RUNG
   RUNG wire#powerrail
      Contact( #Ax_Testa.COut.PlusCheckNext )
   END_RUNG wire#w2
   RUNG wire#powerrail
      Contact( #Ax_Testa.COut.MinusRunning )
      Contact( #Ax_Coda.COut.MinusRunning )
      Coil( #COut.Minus_Running )
   END_RUNG
   RUNG wire#powerrail
      Contact( #Ax_Testa.COut.PlusRunning )
      Contact( #Ax_Coda.COut.PlusRunning )
      Coil( #COut.Plus_Running )
   END_RUNG
   // the same network as SCL:
   #COut.Standstill := #Ax_Testa.Sts.Standstill AND #Ax_Coda.Sts.Standstill;
   #COut.Minus_CheckNext := #Ax_Coda.COut.MinusCheckNext OR #Ax_Testa.COut.MinusCheckNext;
   #COut.Plus_CheckNext := #Ax_Coda.COut.PlusCheckNext OR #Ax_Testa.COut.PlusCheckNext;
   #COut.Minus_Running := #Ax_Testa.COut.MinusRunning AND #Ax_Coda.COut.MinusRunning;
   #COut.Plus_Running := #Ax_Testa.COut.PlusRunning AND #Ax_Coda.COut.PlusRunning;
END_REGION

REGION Network 44: <<< MACHINE STATUS >>>
END_REGION

REGION Network 45: Collect machine to zone interface (internal machines OR)
   RUNG wire#powerrail
      "MachineInterface_2_To_1"(AdditionalAlarms := wire#w1, AdditionalWarnings := wire#w2, MachineInterface_1 := #Ax_Testa.MachineInterface, MachineInterface_2 := #Ax_Coda.MachineInterface, Ret_Val => #MachineInterface)
   END_RUNG
   RUNG wire#powerrail
      I_Contact( #Alarm.CheckBothAxMove )
      Not()
   END_RUNG wire#w1
   RUNG wire#powerrail
      I_Contact( #Warning.MissingCnd.OP_VAI_A_PRELIEVO )
      I_Contact( #Warning.MissingCnd.OP_VAI_A_DEPOSITO )
      Not()
   END_RUNG wire#w2
   // the same network as SCL:
   #MachineInterface := "MachineInterface_2_To_1"(MachineInterface_1 := #Ax_Testa.MachineInterface,
                           MachineInterface_2 := #Ax_Coda.MachineInterface,
                           AdditionalAlarms := NOT (NOT #Alarm.CheckBothAxMove),
                           AdditionalWarnings := NOT (NOT #Warning.MissingCnd.OP_VAI_A_PRELIEVO AND NOT #Warning.MissingCnd.OP_VAI_A_DEPOSITO));
END_REGION
END_FUNCTION_BLOCK
